PROGRAM A23
VAR
	//robot5 : RobotA23;
	//robot6 : RobotA23;
	wrapperA23 : WrapMachine;
END_VAR

METHOD PRIVATE callHardware : BOOL
VAR_INPUT
END_VAR
END_METHOD

METHOD PRIVATE runModules : BOOL
VAR_INPUT
END_VAR
// NETWORK 1
END_METHOD

METHOD PRIVATE setupHardware : BOOL
VAR
	i : INT;
END_VAR
END_METHOD

END_PROGRAM

(* stored: Version 1.1.0.1, ProductVersion 3.1.4024.11
   POU A23: Id {1398fc59-7eb8-4b8a-923a-7c8bc34caf55}, SpecialFunc None
   Method callHardware: Id {0cc553bd-e8cb-4e01-bbeb-d162de020df2}
   Method runModules: Id {391bad03-4ba2-4862-b86e-854fa76dcbef}
   Method setupHardware: Id {a64c747f-a35f-4a39-8af5-03ecfd93413f} *)
